Staubli VAL3: Tester.pjx

--- Tester.pjx ---
Parameters version=s7.11.2 stackSize=5000 millimeterUnit=true
Program file=start.pgx
Program file=stop.pgx
Data file=Tester.dtx

--- Tester.dtx ---
mdesc mNomSpeed
tool tTool = {z=110, fatherId=flange[0], ioLink=valve1}

--- start.pgx ---
program start()
begin
  cls()
  movej(JHome,tTool, mNomSpeed)
  waitEndMove()
  movej(JApproach1,tTool, mNomSpeed)
  waitEndMove()
  do
    // Leo caracter
    clearBuffer(sSioOrdenador)
    delay(5)
    nTest = sioGet(sSioOrdenador, l_nNumero)
    put("Test :")
    put(nTest)
    put(" L_nNumero :")
    put(l_nNumero)
    putln(" ")

    sioSet(sSioOrdenador, l_nNumero)


  until l_nNumero == 13
end
